# EPICS substitutions: TRITON/TRITON-IOC-01App/Db/TRITON_valves.substitutions
file TRITON_valves.template {

pattern {PORT, P, VALVE}
{"\$(PORT)", "\$(P)", "1"}
{"\$(PORT)", "\$(P)", "2"}
{"\$(PORT)", "\$(P)", "3"}
{"\$(PORT)", "\$(P)", "4"}
{"\$(PORT)", "\$(P)", "5"}
{"\$(PORT)", "\$(P)", "6"}
{"\$(PORT)", "\$(P)", "7"}
{"\$(PORT)", "\$(P)", "8"}
{"\$(PORT)", "\$(P)", "9"}
{"\$(PORT)", "\$(P)", "10"}
}
